// Exposes _TaskInfo[x] information for the task index the object is instantied in.
//
// After declaration, each property can be directly accessed.
//
// Set the index using task.Index
FUNCTION_BLOCK T_Task // Simply exposes task information.
VAR
   // Backing Properties
   _index : BYTE := 1;
   _cycleTimeInMs : LREAL;
   _isFirstScan : BOOL;
   _cycleTimeExceeded : BOOL;
   _name : STRING(63);
   _runTimeInMs : UDINT;
   _distributedClockTimeInMs : LINT;
   _distributedClockTimeInNs : LINT;

   // FBs
   initialised : BOOL := FALSE;
   taskIndex : GETCURTASKINDEX;

END_VAR

VAR CONSTANT
   HUNDRED_NS_IN_MS : LINT := 10000;
   NS_IN_MS : LINT := 1000000;
   MS_IN_SECOND : LREAL := 1000.0;
END_VAR

// Number of task cycles executed.
PROPERTY PUBLIC CycleCount : UDINT
GET
cycleCount := TwinCAT_SystemInfoVarList._TaskInfo[_index].CycleCount;
END_GET
END_PROPERTY

// Configured cycles per second (1 / task time)
PROPERTY CyclesPerSecond : LREAL
GET
CyclesPerSecond := 1 / CycleTimeInSecs;
END_GET
END_PROPERTY

// Last cycle time exceeded
PROPERTY CycleTimeExceeded : BOOL
GET
_cycleTimeExceeded := TwinCAT_SystemInfoVarList._TaskInfo[_index].CycleTimeExceeded;
cycleTimeExceeded := _cycleTimeExceeded;
END_GET
END_PROPERTY

// Configured task cycle time in ms
PROPERTY CycleTimeInMs : LREAL
GET
_cycleTimeInMs := TO_LREAL(TwinCAT_SystemInfoVarList._TaskInfo[_index].CycleTime) / LINT_TO_LREAL(HUNDRED_NS_IN_MS); // CycleTime expressed in 100ns units.
cycleTimeInMs := _cycleTimeInMs;
END_GET
END_PROPERTY

// Configured task cycle time in seconds
PROPERTY CycleTimeInSecs : LREAL
GET
CycleTimeInSecs := CycleTimeInMs / MS_IN_SECOND;
END_GET
END_PROPERTY

PROPERTY DateString : STRING
GET
VAR
   temp : STRING;
END_VAR
// remove the trailing time: 2018-07-30_09-23-47
temp := DELETE(TO_STRING(DateTimeString), 9, 11);

// 2018-07-30
DateString := temp;
END_GET
END_PROPERTY

PROPERTY DateTimeFromDc : DATE_AND_TIME
GET
DateTimeFromDc := LINT_TO_DT(TO_LINT(DT#2000-1-1-00:00) + TwinCAT_SystemInfoVarList._TaskInfo[_index].DcTaskTime / 1000000000);
END_GET
END_PROPERTY

PROPERTY DateTimeString : STRING
GET
VAR
   temp : STRING;
END_VAR
// remove the leading DT# : DT#2018-07-30-09:23:47
temp := DELETE(TO_STRING(DateTimeFromDc), 3, 1);
// add underscore between datae and time 2018-07-30-09:23:47
temp := REPLACE(temp, '_', 1, 11);
// replace the colons with dashes 2018-07-30_09:23:47
temp := REPLACE(REPLACE(temp, '-', 1, 14), '-', 1, 17);

// 2018-07-30_09-23-47
DateTimeString := temp;
END_GET
END_PROPERTY

//Distributed clock time in milliseconds.
PROPERTY PUBLIC DistributedClockTimeInMs : LINT
GET
_distributedClockTimeInMs := TwinCAT_SystemInfoVarList._TaskInfo[_index].DcTaskTime / NS_IN_MS; // CycleTime expressed ns.
DistributedClockTimeInMs := _distributedClockTimeInMs;
END_GET
END_PROPERTY

//Distributed clock time in nanoseconds.
PROPERTY PUBLIC DistributedClockTimeInNs : LINT
GET
_distributedClockTimeInNs := TwinCAT_SystemInfoVarList._TaskInfo[_index].DcTaskTime; // CycleTime expressed ns.
DistributedClockTimeInNs := _distributedClockTimeInNs;
END_GET
END_PROPERTY

//Distributed clock time in milliseconds.
PROPERTY PUBLIC DistributedClockTimeInSecs : LINT
GET
DistributedClockTimeInSecs := DistributedClockTimeInMs / 1000;
END_GET
END_PROPERTY

//Get/Set the task for the infomration required. Can use "SetToThisTask()" to set to local task.
PROPERTY PUBLIC Index : BYTE
GET // PUBLIC
Index := _index;
END_GET
SET // PUBLIC
_index := Index;
END_SET
END_PROPERTY

PROPERTY IsFirstScan : BOOL
GET
_isFirstScan := TwinCAT_SystemInfoVarList._TaskInfo[_index].FirstCycle;
IsFirstScan := _isFirstScan;
END_GET
END_PROPERTY

{attribute 'monitoring' := 'call'}
PROPERTY Name : STRING(63)
GET
_name := TwinCAT_SystemInfoVarList._TaskInfo[_index].TaskName;
Name := _name;
END_GET
END_PROPERTY

//set the task object to this task
METHOD PUBLIC SetToThisTask : BOOL
VAR
   curTask : GETCURTASKINDEX;
END_VAR
curTask();
Index := curTask.index;
END_METHOD

PROPERTY TimeString : STRING
GET
VAR
   temp : STRING;
END_VAR
// remove the leading date 2018-07-30_09-23-47
temp := DELETE(TO_STRING(DateTimeString), 11, 1);

// 09-23-47
TimeString := temp;
END_GET
END_PROPERTY

END_FUNCTION_BLOCK

(* stored: Version 1.1.0.1, ProductVersion 3.1.4024.11
   POU T_Task: Id {91408a89-9e5e-4cd9-a531-bed854a04d51}, SpecialFunc None
   Folder Properties: Id {40705766-e38a-4fab-b379-1b30258dfd7b}
   Property CycleCount: Id {6041aa89-f745-4903-948c-e044fe1a39e9}
   Get Get: Id {af07d638-7ccb-41a9-8d1f-19e3538be3a6}
   Property CyclesPerSecond: Id {8e563278-f639-4356-aa4b-c2aadc67d469}
   Get Get: Id {8ba279ac-4db3-4e47-88a6-9987f4f4010d}
   Property CycleTimeExceeded: Id {2dc58f71-ecc5-4281-a35b-f01931a07368}
   Get Get: Id {ba7b93c6-8197-4cca-9c0d-7bcf6c56b937}
   Property CycleTimeInMs: Id {58f2eb2c-ba92-4545-b960-fd1836a8957c}
   Get Get: Id {4fb0f5c0-b166-4fd4-8daa-1e863446cffa}
   Property CycleTimeInSecs: Id {df7cd388-77d1-449a-9343-e24dd5989a77}
   Get Get: Id {f02673c2-dc80-4fe8-9256-f7098f020899}
   Property DateString: Id {616e5652-030b-4cd6-9192-7709b5fd84f8}
   Get Get: Id {0581ed3f-a33f-4c7f-b30d-98f628a4400a}
   Property DateTimeFromDc: Id {59a9e3cb-3f43-4481-8abb-f488ade44dd1}
   Get Get: Id {b0d79845-6ae9-4e73-ae5d-458379ae4868}
   Property DateTimeString: Id {ab8ee405-c790-408e-9600-9288b33b1474}
   Get Get: Id {61ecf890-d2fd-4dcd-9a03-fd6d70e13eda}
   Property DistributedClockTimeInMs: Id {ad308fd0-a973-437e-be58-90470e8ef930}
   Get Get: Id {2d876189-ac67-4e4f-9a27-b4eeaad97533}
   Property DistributedClockTimeInNs: Id {e8e863a3-bf8f-4578-8d3d-d32c7bdfbcd7}
   Get Get: Id {b46378c8-0e1f-4973-9b7f-f91e069d3e26}
   Property DistributedClockTimeInSecs: Id {370d3deb-7b42-403a-9b38-24a446961671}
   Get Get: Id {a29bac17-28db-4ddc-9253-5731fb2ea9b7}
   Property Index: Id {e3f963f0-b880-4563-9015-cbd2aab42b42}
   Get Get: Id {3a6c812c-f41b-414b-abab-4b0101e262da}
   Set Set: Id {56c7d3a0-c8fb-4dd5-b35a-fc3e2d7423a5}
   Property IsFirstScan: Id {1aa53d71-32fb-4f84-86ef-4fa13b3630c5}
   Get Get: Id {9d3a93a4-63a8-463f-9b32-444c5411721f}
   Property Name: Id {58ad3b49-926d-4ebc-8baa-2c23d6ed7d4f}
   Get Get: Id {3997e70e-6fe6-470b-b9d3-da89c8ae110d}
   Method SetToThisTask: Id {5eb1e400-790b-4fee-887d-61c3d51d6183}
   Property TimeString: Id {e1d88600-633d-4a6c-8840-1f294aad9e86}
   Get Get: Id {e50c2d43-b2b8-41d2-9825-b04dca7f3999} *)
